// TIA Portal V20 export
// export: Created 2025-09-14T11:16:00.0000000Z, ExportSetting WithDefaults
VAR_GLOBAL   // PLC tag table "TagTable_AI"
   RTU1_RAT_Temp AT %IW64 : Real;
   RTU1_OAT_Temp AT %IW66 : Real;
   RTU1_DAT_Temp AT %IW68 : Real;
END_VAR
